FUNCTION_BLOCK NumericValue_PHYSA (* Input service interface function block — outputs physical REAL value via AR adapter (wraps NumericValue_PHYS) *)
  (* Standard: ISO 11783-6; Description: Copyright (c) 2026 Meisterschulen am Ostbahnhof This program and the accompanying materials are made available under the terms of the Eclipse Public License 2.0 which is available at https://www.eclipse.org/legal/epl-2.0/ SPDX-License-Identifier: EPL-2.0 *)
  (* Version 1.0, 2026-04-14, Franz Höpfinger, Meisterschulen am Ostbahnhof, initial API and implementation and/or initial documentation *)
  PACKAGE isobus::UT::io::NumericValue;
  IMPORT logiBUS::utils::conversion::phys::NumericObjectPool_S;
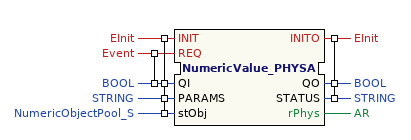
  EVENT_INPUT
    INIT : EInit WITH QI, PARAMS, stObj; (* Service Initialization *)
    REQ WITH QI; (* Service Request *)
  END_EVENT
  EVENT_OUTPUT
    INITO : EInit WITH QO, STATUS; (* Initialization Confirm *)
  END_EVENT
  VAR_INPUT
    QI : BOOL; (* Event Input Qualifier *)
    PARAMS : STRING; (* Service Parameters *)
    stObj : logiBUS::utils::conversion::phys::NumericObjectPool_S; (* Object pool properties (u16ObjId, scale, offset, decimals) *)
  END_VAR
  VAR_OUTPUT
    QO : BOOL; (* Event Output Qualifier *)
    STATUS : STRING; (* Service Status *)
  END_VAR
  PLUGS
    rPhys : adapter::types::unidirectional::AR; (* Physical REAL value output *)
  END_PLUGS
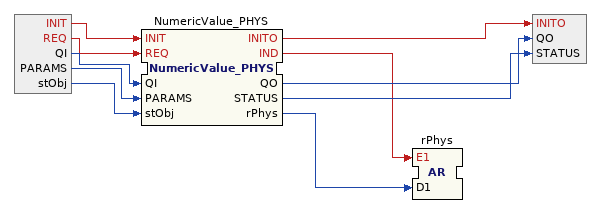
  FBS
    NumericValue_PHYS : isobus::UT::io::NumericValue::NumericValue_PHYS;
  END_FBS
  EVENT_CONNECTIONS
    INIT TO NumericValue_PHYS.INIT;
    REQ TO NumericValue_PHYS.REQ;
    NumericValue_PHYS.INITO TO INITO;
    NumericValue_PHYS.IND TO rPhys.E1;
  END_CONNECTIONS
  DATA_CONNECTIONS
    stObj TO NumericValue_PHYS.stObj;
    PARAMS TO NumericValue_PHYS.PARAMS;
    QI TO NumericValue_PHYS.QI;
    NumericValue_PHYS.QO TO QO;
    NumericValue_PHYS.STATUS TO STATUS;
    NumericValue_PHYS.rPhys TO rPhys.D1;
  END_CONNECTIONS
END_FUNCTION_BLOCK
